FUNCTION_BLOCK FB_NOTT_TipTilt
VAR
//	Tip Actuators A 

	NTPA1:			FB_MOTOR;
	NTPA2:			FB_MOTOR;
	NTPA3:			FB_MOTOR;
	NTPA4:			FB_MOTOR;
	
	ptrTipActuatorsA:	ARRAY [1..4] OF POINTER TO FB_MOTOR;
	// GUI stuff
	guiTipActuatorsAIndex:	UINT := 1;	// Index for Tip Actuators A Engineering GUI

//	Tilt Actuators A 
	
	NTTA1:			FB_MOTOR;
	NTTA2:			FB_MOTOR;
	NTTA3:			FB_MOTOR;
	NTTA4:			FB_MOTOR;
	
	ptrTiltActuatorsA:	ARRAY [1..4] OF POINTER TO FB_MOTOR;
	// GUI stuff
	guiTiltActuatorsAIndex:	UINT := 1;	// Index for Tilt Actuators A Engineering GUI	
	
//	Tip Actuators B 

	NTPB1:			FB_MOTOR;
	NTPB2:			FB_MOTOR;
	NTPB3:			FB_MOTOR;
	NTPB4:			FB_MOTOR;
	
	ptrTipActuatorsB:	ARRAY [1..4] OF POINTER TO FB_MOTOR;
	// GUI stuff
	guiTipActuatorsBIndex:	UINT := 1;	// Index for Tip Actuators B Engineering GUI	

//	Tilt Actuators B 
	
	NTTB1:			FB_MOTOR;
	NTTB2:			FB_MOTOR;
	NTTB3:			FB_MOTOR;
	NTTB4:			FB_MOTOR;
	
	ptrTiltActuatorsB:	ARRAY [1..4] OF POINTER TO FB_MOTOR;
	// GUI stuff
	guiTiltActuatorsBIndex:	UINT := 1;	// Index for Tilt Actuators A Engineering GUI

// Simulation

//	Sim Tip Actuators A 

	SIM_NTPA1:			FB_SIM_MOTOR;
	SIM_NTPA2:			FB_SIM_MOTOR;
	SIM_NTPA3:			FB_SIM_MOTOR;
	SIM_NTPA4:			FB_SIM_MOTOR;

//	Sim Tilt Actuators A 
	
	SIM_NTTA1:			FB_SIM_MOTOR;
	SIM_NTTA2:			FB_SIM_MOTOR;
	SIM_NTTA3:			FB_SIM_MOTOR;
	SIM_NTTA4:			FB_SIM_MOTOR;
	
//	Sim Tip Actuators B 

	SIM_NTPB1:			FB_SIM_MOTOR;
	SIM_NTPB2:			FB_SIM_MOTOR;
	SIM_NTPB3:			FB_SIM_MOTOR;
	SIM_NTPB4:			FB_SIM_MOTOR;
		

//	Sim Tilt Actuators B 
	
	SIM_NTTB1:			FB_SIM_MOTOR;
	SIM_NTTB2:			FB_SIM_MOTOR;
	SIM_NTTB3:			FB_SIM_MOTOR;
	SIM_NTTB4:			FB_SIM_MOTOR;	
	
END_VAR

M_Configure();

//	Tip Actuators A 

NTPA1(
	in_bSafe:= , 
	in_bDisableIfUnsafe:= , 
	sName:= 'NTPA1', 
	nNOVRAM_DevId:= 6, 
	nNOVRAM_Offset:= 5000);
	
NTPA2(
	in_bSafe:= , 
	in_bDisableIfUnsafe:= , 
	sName:= 'NTPA2', 
	nNOVRAM_DevId:= 6, 
	nNOVRAM_Offset:= 6000);
	
NTPA3(
	in_bSafe:= , 
	in_bDisableIfUnsafe:= , 
	sName:= 'NTPA3', 
	nNOVRAM_DevId:= 6, 
	nNOVRAM_Offset:= 7000);
	
NTPA4(
	in_bSafe:= , 
	in_bDisableIfUnsafe:= , 
	sName:= 'NTPA4', 
	nNOVRAM_DevId:= 6, 
	nNOVRAM_Offset:= 8000);
	
//	Tilt Actuators A
	
NTTA1(
	in_bSafe:= , 
	in_bDisableIfUnsafe:= , 
	sName:= 'NTTA1', 
	nNOVRAM_DevId:= 6, 
	nNOVRAM_Offset:= 9000);
	
NTTA2(
	in_bSafe:= , 
	in_bDisableIfUnsafe:= , 
	sName:= 'NTTA2', 
	nNOVRAM_DevId:= 6, 
	nNOVRAM_Offset:= 10000);
	
NTTA3(
	in_bSafe:= , 
	in_bDisableIfUnsafe:= , 
	sName:= 'NTTA3', 
	nNOVRAM_DevId:= 6, 
	nNOVRAM_Offset:= 11000);
	
NTTA4(
	in_bSafe:= , 
	in_bDisableIfUnsafe:= , 
	sName:= 'NTTA4', 
	nNOVRAM_DevId:= 6, 
	nNOVRAM_Offset:= 12000);
	
//	Tip Actuators B

NTPB1(
	in_bSafe:= , 
	in_bDisableIfUnsafe:= , 
	sName:= 'NTPB1', 
	nNOVRAM_DevId:= 6, 
	nNOVRAM_Offset:= 13000);
	
NTPB2(
	in_bSafe:= , 
	in_bDisableIfUnsafe:= , 
	sName:= 'NTPB2', 
	nNOVRAM_DevId:= 6, 
	nNOVRAM_Offset:= 14000);
	
NTPB3(
	in_bSafe:= , 
	in_bDisableIfUnsafe:= , 
	sName:= 'NTPB3', 
	nNOVRAM_DevId:= 6, 
	nNOVRAM_Offset:= 15000);
	
NTPB4(
	in_bSafe:= , 
	in_bDisableIfUnsafe:= , 
	sName:= 'NTPB4', 
	nNOVRAM_DevId:= 6, 
	nNOVRAM_Offset:= 16000);

//	Tilt Actuators B 

NTTB1(
	in_bSafe:= , 
	in_bDisableIfUnsafe:= , 
	sName:= 'NTTB1', 
	nNOVRAM_DevId:= 6, 
	nNOVRAM_Offset:= 17000);
	
NTTB2(
	in_bSafe:= , 
	in_bDisableIfUnsafe:= , 
	sName:= 'NTTB2', 
	nNOVRAM_DevId:= 6, 
	nNOVRAM_Offset:= 18000);
	
NTTB3(
	in_bSafe:= , 
	in_bDisableIfUnsafe:= , 
	sName:= 'NTTB3', 
	nNOVRAM_DevId:= 6, 
	nNOVRAM_Offset:= 19000);
	
NTTB4(
	in_bSafe:= , 
	in_bDisableIfUnsafe:= , 
	sName:= 'NTTB4', 
	nNOVRAM_DevId:= 6, 
	nNOVRAM_Offset:= 20000);

// Simulation

SIM_NTPA1(ptrCfg:= ADR(NTPA1.cfg), ptrStat:= ADR(NTPA1.stat));
SIM_NTPA2(ptrCfg:= ADR(NTPA2.cfg), ptrStat:= ADR(NTPA2.stat));
SIM_NTPA3(ptrCfg:= ADR(NTPA3.cfg), ptrStat:= ADR(NTPA3.stat));
SIM_NTPA4(ptrCfg:= ADR(NTPA4.cfg), ptrStat:= ADR(NTPA4.stat));

SIM_NTPB1(ptrCfg:= ADR(NTPB1.cfg), ptrStat:= ADR(NTPB1.stat));
SIM_NTPB2(ptrCfg:= ADR(NTPB2.cfg), ptrStat:= ADR(NTPB2.stat));
SIM_NTPB3(ptrCfg:= ADR(NTPB3.cfg), ptrStat:= ADR(NTPB3.stat));
SIM_NTPB4(ptrCfg:= ADR(NTPB4.cfg), ptrStat:= ADR(NTPB4.stat));

SIM_NTTA1(ptrCfg:= ADR(NTTA1.cfg), ptrStat:= ADR(NTTA1.stat));
SIM_NTTA2(ptrCfg:= ADR(NTTA2.cfg), ptrStat:= ADR(NTTA2.stat));
SIM_NTTA3(ptrCfg:= ADR(NTTA3.cfg), ptrStat:= ADR(NTTA3.stat));
SIM_NTTA4(ptrCfg:= ADR(NTTA4.cfg), ptrStat:= ADR(NTTA4.stat));

SIM_NTTB1(ptrCfg:= ADR(NTTB1.cfg), ptrStat:= ADR(NTTB1.stat));
SIM_NTTB2(ptrCfg:= ADR(NTTB2.cfg), ptrStat:= ADR(NTTB2.stat));
SIM_NTTB3(ptrCfg:= ADR(NTTB3.cfg), ptrStat:= ADR(NTTB3.stat));
SIM_NTTB4(ptrCfg:= ADR(NTTB4.cfg), ptrStat:= ADR(NTTB4.stat));

METHOD M_Configure : BOOL
VAR_INPUT
END_VAR
//	Tip Actuators A 

ptrTipActuatorsA[1] := ADR(NTPA1);
ptrTipActuatorsA[2] := ADR(NTPA2);
ptrTipActuatorsA[3] := ADR(NTPA3);
ptrTipActuatorsA[4] := ADR(NTPA4);

//	Tilt Actuators A 

ptrTiltActuatorsA[1] := ADR(NTTA1);
ptrTiltActuatorsA[2] := ADR(NTTA2);
ptrTiltActuatorsA[3] := ADR(NTTA3);
ptrTiltActuatorsA[4] := ADR(NTTA4);

//	Tip Actuators B

ptrTipActuatorsB[1] := ADR(NTPB1);
ptrTipActuatorsB[2] := ADR(NTPB2);
ptrTipActuatorsB[3] := ADR(NTPB3);
ptrTipActuatorsB[4] := ADR(NTPB4);

//	Tilt Actuators B

ptrTiltActuatorsB[1] := ADR(NTTB1);
ptrTiltActuatorsB[2] := ADR(NTTB2);
ptrTiltActuatorsB[3] := ADR(NTTB3);
ptrTiltActuatorsB[4] := ADR(NTTB4);
END_METHOD

END_FUNCTION_BLOCK

(* stored: Version 1.1.0.1, ProductVersion 3.1.4024.12
   POU FB_NOTT_TipTilt: Id {f38a4431-261f-431d-a596-42067753e201}, SpecialFunc None
   Method M_Configure: Id {08fcbaf5-ced8-4250-a494-ef908cd2e0a2} *)
